# EPICS StreamDevice protocol: protocols/hudp.proto
Terminator = LF;
ExtraInput = Ignore;

getIp {
	out "ip";
	in "%s";
}

getDstIp {
	out "dst_ip";
	in "%s";
}

getDstPort {
	out "dst_port";
	in "%d";
}

getTxPktSz {
	out "tx_pkt_sz";
	in "%d";
}

getRxSrcIp {
	out "rx_src_ip";
	in "%s";
}

getRxPort {
	out "rx_port";
	in "%d";
}

getCtrl {
	out "ctrl";
	in "%d";
}

setCtrl {
	out "ctrl %d";
	in "";
}
